// Writes a float field value, without a tag, to the stream.
FUNCTION F_WriteFloat : HRESULT
VAR_IN_OUT
    aBuffer : ARRAY [*] OF BYTE;
    stState : ST_WriterInternalState;
END_VAR
VAR_INPUT CONSTANT
    fValue : REAL;
END_VAR
VAR CONSTANT
    cLength : UDINT := SIZEOF(fValue);
END_VAR
VAR
    fTmp : REAL;
END_VAR


F_WriteFloat := S_OK;

IF stState.nBufferSize - stState.nBufferPos < cLength THEN
    F_WriteFloat := stState.eWriterErrorCode := E_WriterErrorCode.TruncatedMessage;
    stState.bError := TRUE;
    RETURN;
END_IF
{warning 'TODO: Check for endianess?'}
fTmp := fValue;

MEMCPY(destAddr:= ADR(aBuffer[stState.nBufferPos]), srcAddr:= ADR(fTmp), n:= cLength);

END_FUNCTION

(* stored: Version 1.1.0.1
   POU F_WriteFloat: Id {31c0f91b-2323-44ae-b077-dd782051d522}, SpecialFunc None *)
